FUNCTION_BLOCK FB_MovingAverageReal
VAR_INPUT
	// Value to add to the moving average.
	ValueToAdd : LREAL;
	// The number of values to store in the array.
	NumValuesToUse : UINT := TO_UINT(UPPER_BOUND(AverageArray, 1) - LOWER_BOUND(AverageArray, 1) + 1);
END_VAR
VAR_IN_OUT
	AverageArray  : ARRAY [*] OF LREAL;
END_VAR
VAR_OUTPUT
	CurrentValue : LREAL;
END_VAR
VAR
	CurrentIndex : UINT;
	NumValuesAdded: UINT;
END_VAR
VAR_TEMP
	Counted : UINT;
	I: DINT;
	Sum: LREAL;
	ArrayLength : UINT := TO_UINT(UPPER_BOUND(AverageArray, 1) - LOWER_BOUND(AverageArray, 1) + 1);
END_VAR

// Compute average over array.
// The order of this addition and MOD are important to avoid going out of bounds.
NumValuesToUse := MIN(ArrayLength, NumValuesToUse);
AverageArray[CurrentIndex] := ValueToAdd;
CurrentIndex := CurrentIndex + 1;
CurrentIndex := CurrentIndex MOD NumValuesToUse;
NumValuesAdded := MIN(NumValuesAdded + 1 , NumValuesToUse);
IF NumValuesAdded > 0 THEN
	FOR I := LOWER_BOUND(AverageArray, 1) TO UPPER_BOUND(AverageArray, 1) BY 1 DO
		Sum := Sum + AverageArray[I];
		Counted := Counted + 1;
		// Don't count more than the number of values.
		IF Counted > NumValuesAdded THEN
			EXIT;
		END_IF
	END_FOR
END_IF
CurrentValue := TO_REAL(Sum / NumValuesAdded);

END_FUNCTION_BLOCK

(* stored: Version 1.1.0.1, ProductVersion 3.1.4022.16
   POU FB_MovingAverageReal: Id {fda7e211-5c6c-492f-ac36-81cea3ee5c49}, SpecialFunc None *)
